// TIA Portal V20 export
DATA_BLOCK "COLLECTIVE_SIGNAL_DB"   // DB117
{ S7_Optimized_Access := 'TRUE' }
// stored: MemoryReserve 100
   VAR
      COLLECTIVE_PD_ALARM : Bool;   // Collective signal: Alarms / Sammelsignal: Alarme
      COLLECTIVE_PD_WARNING : Bool;   // Collective signal: Warning / Sammelsignal: Warnungen
      COLLECTIVE_PD_INFO : Bool;   // Collective signal: Information / Sammelsignal: Information / Sammelsignal: 信息
      COLLECTIVE_SIGNAL_PD : USInt;   // 1: Alarm, 2: Warnung, 3: Information / 1: Alarm, 2: Warning, 3: Information / 1: 警报, 2: 警告, 3: 信息
   END_VAR
BEGIN
END_DATA_BLOCK
